PROGRAM P_ScadaAlarmsMapping
VAR
		i: UINT;
END_VAR


FOR i := 1 TO iMaxAlarms DO

	arrScadaAlarms[i].b := BOOL_TO_INT ( arrAlarms[i].b );

END_FOR

END_PROGRAM

(* stored: Version 1.1.0.1, ProductVersion 3.1.4024.9
   POU P_ScadaAlarmsMapping: Id {b07e35a5-255d-4329-8314-96e0e17ff707}, SpecialFunc None *)
